	1:	
		sError															:= '';
		bPreCheckDone													:= FALSE;
		P_M01_RS01.close_valves											:= P_M01.bRS01;
		P_M01_RS02.close_valves											:= P_M01.bRS02;
		P_M01_RS03.close_valves											:= P_M01.bRS03;
		P_M01_RS01.retract_all_clamps									:= P_M01.bRS01;
		P_M01_RS02.retract_all_clamps									:= P_M01.bRS02;
		P_M01_RS03.retract_all_clamps									:= P_M01.bRS03;
		rTime															:= _VALVE_TIME;
		iAxStep															:= iAxStep + 1;
	
	2:	
		bTimer															:= TRUE;
		bPass1															:= (P_M01.bRS01 AND P_M01_RS01.R_S.valves_clear AND m01_rs1.steam_control_valve_position < _VALVE_CLOSED) OR NOT P_M01.bRS01;
		bPass2															:= (P_M01.bRS02 AND P_M01_RS02.R_S.valves_clear AND m01_rs2.steam_control_valve_position < _VALVE_CLOSED) OR NOT P_M01.bRS02;
		bPass3															:= (P_M01.bRS03 AND P_M01_RS03.R_S.valves_clear AND m01_rs3.steam_control_valve_position < _VALVE_CLOSED) OR NOT P_M01.bRS03;
		IF bPass1 AND bPass2 AND bPass3 THEN
			bTimer														:= FALSE;
			iAxStep														:= iAxStep + 1;
		ELSIF tonTimer.Q THEN
			sError														:= 'Valve Error';
			iAxStep														:= 99;
		END_IF

	3:
		IF (P_M01_RS01.inlet_air_high_temp_count + P_M01_RS02.inlet_air_high_temp_count + P_M01_RS03.inlet_air_high_temp_count) <= _HIGH_CART_READINGS_MAX THEN
			iAxStep														:= iAxStep + 1;
		ELSE
			sError														:= gsHighTempCountError;
			iAxStep														:= 99;
		END_IF

	4:
		bPass1															:= (P_M01.bRS01 AND P_M01_RS01.R_S.all_clamps_retracted) OR NOT P_M01.bRS01; 
		bPass2															:= (P_M01.bRS02 AND P_M01_RS02.R_S.all_clamps_retracted) OR NOT P_M01.bRS02; 
		bPass3															:= (P_M01.bRS03 AND P_M01_RS03.R_S.all_clamps_retracted) OR NOT P_M01.bRS03; 
		IF bPass1 AND bPass2 AND bPass3 THEN
			iAxStep														:= iAxStep + 1;
		ELSE
			sError														:= gsClampRetractError;
			iAxStep														:= 99;
		END_IF
		
	5:
		IF NOT u.os_air_unsafe_temp THEN
			iAxStep														:= iAxStep + 1;
		ELSE
			sError														:= gsInletAirTempRangeError;
			iAxStep														:= 99;
		END_IF
		
	6:
		bPass1															:= (P_M01.bRS01 AND P_M01_RS01.average_pressure_within_ambient) OR NOT P_M01.bRS01;
		bPass2															:= (P_M01.bRS02 AND P_M01_RS02.average_pressure_within_ambient) OR NOT P_M01.bRS02;
		bPass3															:= (P_M01.bRS03 AND P_M01_RS03.average_pressure_within_ambient) OR NOT P_M01.bRS03;
		IF NOT bPass1 OR NOT bPass2 OR NOT bPass3 THEN
			sError														:=  gsAmbientPressureError;
		END_IF
		iAxStep															:= 99;
		
	99:
		bTimer															:= FALSE;
		bPreCheckDone													:= TRUE;
		iAxStep															:= 0;
				
END_CASE
END_ACTION

METHOD M_Repres_Valve_Error : STRING
VAR_INPUT
END_VAR
VAR
	sErr																: STRING	:= '';
END_VAR
// Phase 0 - P_U01.M_Repres_Valve_Error
// Rev 1.0 - March 12, 2024

IF P_M01.bRS03 THEN
	;//sErr																:= SEL(P_M01_RS03_R4.bRepresValveClear, CONCAT(_RS03, _R4), sErr);
	//sErr																:= SEL(P_M01_RS03_R3.bRepresValveClear, CONCAT(_RS03, _R3), sErr);
	//sErr																:= SEL(P_M01_RS03_R2.bRepresValveClear, CONCAT(_RS03, _R2), sErr);
	//sErr																:= SEL(P_M01_RS03_R1.bRepresValveClear, CONCAT(_RS03, _R1), sErr);
END_IF                                                                                                                                   
IF P_M01.bRS02 THEN                                                                                                                       
	;//sErr																:= SEL(P_M01_RS02_R4.bRepresValveClear, CONCAT(_RS02, _R4), sErr);
	//sErr																:= SEL(P_M01_RS02_R3.bRepresValveClear, CONCAT(_RS02, _R3), sErr);
	//sErr																:= SEL(P_M01_RS02_R2.bRepresValveClear, CONCAT(_RS02, _R2), sErr);
	//sErr																:= SEL(P_M01_RS02_R1.bRepresValveClear, CONCAT(_RS02, _R1), sErr);
END_IF                                                                                                                                   
IF P_M01.bRS01 THEN                                                                                                                       
	//sErr																:= SEL(P_M01_RS01_R4.bRepresValveClear, CONCAT(_RS01, _R4), sErr);
	//sErr																:= SEL(P_M01_RS01_R3.bRepresValveClear, CONCAT(_RS01, _R3), sErr);
	//sErr																:= SEL(P_M01_RS01_R2.bRepresValveClear, CONCAT(_RS01, _R2), sErr);
	//sErr																:= SEL(P_M01_RS01.repres_valves_clear, CONCAT(_RS01, _R1), sErr);
END_IF
M_Repres_Valve_Error													:= SEL(sErr <> '', sErr, CONCAT(sErr, gsRepressurizationValveError));
END_METHOD

END_PROGRAM

(* stored: Version 1.1.0.1, ProductVersion 3.1.4024.12
   POU P_U01: Id {dcf8449b-3592-47e4-a482-48f13716f004}, SpecialFunc None
   Action A_BOP_Estop: Id {5c5d44f9-58ec-48e1-911e-c5376b4fba9d}
   Action A_Drains: Id {ab317b0b-7a30-41e9-b5c6-59249957db4c}
   Action A_IO_Points: Id {d2567efd-8816-46e7-a69d-41abdef6a01f}
   Action A_Totalizers: Id {5628a577-b91b-468f-9d37-381d8cfc29f4}
   Action A_Weather_Station: Id {97e557fc-0646-468d-b78c-428d62b1eadb}
   Action A2_WarmUp: Id {3e02c609-752d-4440-9a0e-94c91ce7baf7}
   Action A3_Steam_Bypass: Id {73856173-8e49-4891-b8be-3c57dfbf2633}
   Action A8_Shutdown: Id {dceaad34-9fba-494d-9502-9d4c836ba12b}
   Action A9_Pressure_Drop_Test: Id {b8bf7e66-dcdb-4668-8218-16ff48a3e793}
   Action Ax_Process_Pre_Check: Id {d59aaf0d-9d27-45c8-bc13-c9bb5b8aaff8}
   Method M_Repres_Valve_Error: Id {83f36fa0-ccb5-4077-b38d-3796cb92f31f} *)
